TYPE T_Ctrl_SIf_SLB_In :
STRUCT
END_STRUCT
END_TYPE

(* stored: Version 1.1.0.1, ProductVersion 3.1.0.19
   DUT T_Ctrl_SIf_SLB_In: Id {704f496f-495d-42a5-89ff-7357d38e79d3} *)
